// TIA Portal project "Sensor 1" (V15)

(* hardware
DEVICE "S7-1200 station_1"  S7-1200 Station
   slot 0: "Rack_0"  S7-1200 Rack  Rack  V1.0
   slot 1: "PLC_1"  CPU 1212C AC/DC/Rly  6ES7 212-1BE31-0XB0  V3.0
*)

// ===== PLC "PLC_1"  CPU 1212C AC/DC/Rly =====

VAR_GLOBAL   // PLC tag table "Default tag table"
   "start" AT %I0.0 : Bool;
   "X  marker 1" AT %M0.0 : Bool;
   "stop" AT %I0.2 : Bool;
   "MOTOR 1" AT %Q0.0 : Bool;
   "Sensor" AT %I0.3 : Bool;
   "Sensor marker" AT %M0.2 : Bool;
   "marker 2" AT %M1.1 : Bool;
END_VAR

// folder: System blocks/Program resources

DATA_BLOCK "T1"   // DB1
{ S7_Optimized_Access := 'TRUE' }
AUTHOR : Simatic
FAMILY : IEC
NAME : IEC_TMR
VERSION : 1.0
// stored: InstanceOfName IEC_TIMER
"IEC_TIMER"
BEGIN
END_DATA_BLOCK

// folder: (top level)

ORGANIZATION_BLOCK "Main"   // OB1, LAD, ProgramCycle
TITLE = "Main Program Sweep (Cycle)"
{ S7_Optimized_Access := 'TRUE' }
VERSION : 0.1
BEGIN

REGION Network 1: m0.0
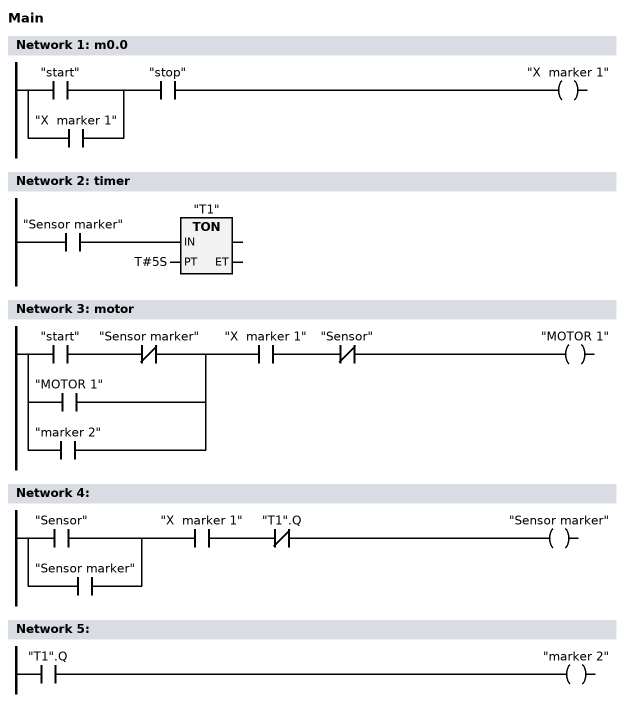
   RUNG wire#powerrail
      Contact( "start" )
      wire#w1
      Contact( "stop" )
      Coil( "X  marker 1" )
   END_RUNG
   RUNG wire#powerrail
      Contact( "X  marker 1" )
   END_RUNG wire#w1
   // the same network as SCL:
   "X  marker 1" := ("start" OR "X  marker 1") AND "stop";
END_REGION

REGION Network 2: timer
   "T1".TON(IN := "Sensor marker", PT := T#5S);
END_REGION

REGION Network 3: motor
   RUNG wire#powerrail
      Contact( "start" )
      I_Contact( "Sensor marker" )
      wire#w1
      Contact( "X  marker 1" )
      I_Contact( "Sensor" )
      Coil( "MOTOR 1" )
   END_RUNG
   RUNG wire#powerrail
      Contact( "MOTOR 1" )
   END_RUNG wire#w1
   RUNG wire#powerrail
      Contact( "marker 2" )
   END_RUNG wire#w1
   // the same network as SCL:
   "MOTOR 1" := (("start" AND NOT "Sensor marker") OR "MOTOR 1" OR "marker 2") AND "X  marker 1" AND NOT "Sensor";
END_REGION

REGION Network 4
   RUNG wire#powerrail
      Contact( "Sensor" )
      wire#w1
      Contact( "X  marker 1" )
      I_Contact( "T1".Q )
      Coil( "Sensor marker" )
   END_RUNG
   RUNG wire#powerrail
      Contact( "Sensor marker" )
   END_RUNG wire#w1
   // the same network as SCL:
   "Sensor marker" := ("Sensor" OR "Sensor marker") AND "X  marker 1" AND NOT "T1".Q;
END_REGION

REGION Network 5
   RUNG wire#powerrail
      Contact( "T1".Q )
      Coil( "marker 2" )
   END_RUNG
   // the same network as SCL:
   "marker 2" := "T1".Q;
END_REGION
END_ORGANIZATION_BLOCK